FUNCTION "Conveer26FO" : Void
{ S7_Optimized_Access := 'FALSE' }
VERSION : 0.1
   VAR_TEMP
      run : Bool;
      error : Bool;
      form : Bool;
      formLeft : Bool;
      formRight : Bool;
      sensorCount : Bool;
      sensorBrake : Bool;
      Brake : Bool;
      workRight : Bool;
      workLeft : Bool;
      FlowLeft : Bool;
      cutoff : Bool;
      "counter" : Int;
      quantityLeft : Int;
      quantityRight : Int;
      stop_box_time : Time;
   END_VAR


BEGIN
	//2 линия
	//"FA26_1_auto_start" := TRUE;//двигатель транспортера в автомате работает

	// "IEC_Timer_28tr_DB".TON(IN:=#sensorBrake,
	//                         PT:=T#3s,
	//                         Q=>#Brake,
	//                         ET=>#stop_box_time);

	IF "Auto3" THEN
	    "KA26_2" := "Robot16".FDO01;//сброс елеватора по команде робота "забрал"
	    "Robot16".TDI01 := "SW26_1";//готово от елеватора роботу
	END_IF;




	IF "SW26_1" AND NOT "Tag_2"//фронт команды забрали
	    OR "Robot16".FDO11 //или закончил сбор паллеты
	THEN//меняем уставку счетчика по сигналам робота "разверни" и "забрал"
	    IF "Robot16".FDO23 //если крайний то по 3
	        AND "Auto3"
	    THEN
	       "KA26_3" := FALSE;//слои
	        "KA26_4" := TRUE;//слои
	        "m301_0" := FALSE;
	        "m301_1" := tRUE;

	    ELSE
	        "KA26_3" := TRUE;//слои
	        "KA26_4" := TRUE;//слои
	        "m301_0" := TRUE;
	        "m301_1" := tRUE;

	    END_IF;
	END_IF;

	"Tag_2" := "SW26_1";

	    IF "Manual3" OR "HalfManual3" THEN
	    "KA26_3" := "m301_0";//слои
	    "KA26_4" := "m301_1";//слои
	END_IF;


	IF "Auto3" THEN
	    "KA26_1" := TRUE;//элеватор пуск
	END_IF;
	//"DB_Counters".SW26.GEAR := TRUE;
	//"DB_Counters".SW26.SP := 4;
	//"DB_Counters".SW26.RESET := FALSE;

	//"00_CounterInteger"(DB_Counter:= "DB_Counters",
	//                     FirstByte:= 36,
	//                     SetValue:= "DB_Counters".SW26.SP,
	//                     Count:= "SW26.1",
	//                     ValueIncrement:= 1,
	//                     CountCurrent:= "DB_Counters".SW26.ACT);


	//"KA26_1" := "SW26_2";
	//IF "DB_Counters".SW26.SET_OK THEN
	//    "KA26_1" := TRUE;
	//END_IF;


	// CASE "Conveer_status"."28_step" OF//db6.dbw0
	//     0://стоп


	//         IF "SW3_1"= FALSE AND "SW3_3" = FALSE THEN //если на входе нет коробок
	//             "Conveer_status"."28_step":=10;
	//         END_IF;
	//         IF "SW3_1" = TRUE AND "SW3_3" = FALSE THEN //если на входе есть коробки
	//             "Conveer_status"."28_step" := 20;
	//         END_IF;

	//         ;
	//     10://нет на входе



	//         IF "SW3_1" = TRUE AND "Robot12".FDO03 = TRUE THEN //если на входе есть коробки
	//             "Conveer_status"."28_step" := 20;
	//         END_IF;

	//         ;
	//     20://есть на входе и не готово



	//         IF "SW3_1"= TRUE AND "SW3_3" = FALSE AND "Robot12".FDO11 = TRUE THEN
	//             //если стопор чегото там
	//             "Conveer_status"."28_step" := 30;
	//         END_IF;

	//         ;
	//     30://загружаем



	//         IF "SW3_3" = TRUE THEN //если  счетчик досчитал
	//             "Conveer_status"."28_step" := 40;
	//         END_IF;
	//         ;
	//     40://подсчет и проверка



	//         IF "SW3_3" = TRUE THEN //если  проверка успешна
	//             "Conveer_status"."28_step" := 50;
	//         END_IF;

	//         ;
	//     50://выполненно


	//         IF "SW3_4" = FALSE OR "SW3_3" = FALSE THEN //если кара то она забирает паллету
	//             "Conveer_status"."28_step" := 0;// не будем ждать пока заберут, робота нужно обслуживать
	//         END_IF;

	//         ;
	//     60://забирают


	//         IF "SW3_4" = TRUE OR "SW3_3" = FALSE OR "SW3_1" = TRUE THEN //если кара или забрали или поставили то
	//             "Conveer_status"."28_step" := 0;
	//         END_IF;

	//         ;

	//     70://возврата нет
	//                "Conveer_status"."28_step" := 0;
	//         ;

	//         ;
	//     ELSE:
	//         ;
	// END_CASE;

END_FUNCTION

